Staubli VAL3: link_it.pgx

public program link_it(string x_sName)
begin
  // link all the point
  call link_all(x_sName)
  // put the base config
  tTraj[x_sName].tData[1].tSuper.toStop=true
  tTraj[x_sName].tData[0].tSuper.moveType=1
  tTraj[x_sName].tData[1].tSuper.moveType=1
  tTraj[x_sName].tData[2].tSuper.moveType=1
  tTraj[x_sName].tData[0].nType=0
  tTraj[x_sName].tData[1].nType=1
  tTraj[x_sName].tData[2].nType=2
  tTraj[x_sName].tData[0].tSuper.comment="appro"
  tTraj[x_sName].tData[1].tSuper.comment="point"
  tTraj[x_sName].tData[2].tSuper.comment="depart"
end
